FUNCTION_BLOCK Sequence1Task_2 EXTENDS TcoCore.TcoTask
VAR_INPUT
    Sequence : TcoCore.ITcoSequencer;
END_VAR

(*~
    <docu>
        <summary>
            Restores this instance to the Ready state. Can be called explicitly or from within one of the restore mechanisms.
            <para>
                See also <see cref="PlcDocu.TcoCore.TcoTask.AutoRestorable()"/>
            </para>
        </summary>
    </docu>
~*)
METHOD Restore : ITcoRestorable
SUPER^.Restore();
THIS^.Sequence.Restore();
END_METHOD

END_FUNCTION_BLOCK

(* stored: Version 1.1.0.1, ProductVersion 3.1.4024.12
   POU Sequence1Task_2: Id {8ac1760f-5fd8-05ef-1ab5-4385a4fb8953}, SpecialFunc None
   Method Restore: Id {07c48c33-290d-0957-0a69-aaec534ba2ef} *)
